TYPE typeMessageRow :
STRUCT
	msgText: STRING(255);
	isAlarm: BOOL; //red
	isWarning: BOOL; //yellow



END_STRUCT
END_TYPE

(* stored: Version 1.1.0.1, ProductVersion 3.1.4024.12
   DUT typeMessageRow: Id {5687a184-79ff-414c-81b1-ad6a2c08ed77} *)
